Yaskawa INFORM job: WEAVING.JBI

/JOB
//NAME WEAVING
//POS
///NPOS 0,0,0,0,0,0
//INST
///DATE 2025/03/03 11:23
///ATTR SC,RW,MC
///GROUP1 RB1
///LVARS 5,5,5,5,0,0,0,0
NOP
GETARG LR000 IARG#(1)
GETARG LR001 IARG#(2)
GETARG LR002 IARG#(3)
MUL LR000 10
MUL LR001 10
MUL LR002 10
SET D080 LR000
SET D081 LR001
SET D082 LR002
END
